INTERFACE I_EventGroupItem

METHOD PUBLIC AddHandler
VAR_INPUT
	EventHandler : I_EventHandler;
END_VAR
END_METHOD

METHOD PUBLIC Dispose
VAR_INPUT
END_VAR
END_METHOD

METHOD PUBLIC Emit
VAR_INPUT
	Event : I_Event;
END_VAR
END_METHOD

METHOD EqualTo : BOOL
VAR_INPUT
	Name : T_MAXSTRING;
END_VAR
END_METHOD

PROPERTY HasHandlers : BOOL
GET
END_GET
END_PROPERTY

PROPERTY PUBLIC Next : I_EventGroupItem
GET
END_GET
SET
END_SET
END_PROPERTY

PROPERTY PUBLIC Previous : I_EventGroupItem
GET
END_GET
SET
END_SET
END_PROPERTY

METHOD RemoveHandler
VAR_INPUT
	EventHandler : I_EventHandler;
END_VAR
END_METHOD

END_INTERFACE

(* stored: Version 1.1.0.1, ProductVersion 3.1.4024.12
   Itf I_EventGroupItem: Id {7a1aa493-2557-41cb-abb3-c16bd9197aae}
   Method AddHandler: Id {23b0f7b4-8051-4dc6-b2fb-d9f1a5f6af37}
   Method Dispose: Id {1d9a84c7-e06c-4aa0-b10a-8120bf170ab4}
   Method Emit: Id {057fcb02-01ee-4f3e-b199-c01963cdefe8}
   Method EqualTo: Id {a0733ef6-95ca-4a6b-b85f-8b85d11ec1e1}
   Property HasHandlers: Id {1d0156d6-948d-4c09-9e8c-940fdf299838}
   Get Get: Id {f93f0960-7100-4f32-804b-08f516727210}
   Property Next: Id {9f8ae168-7fea-40e1-8194-bd7be4b40641}
   Get Get: Id {b1fb12e4-77d8-403f-b6bc-1a0b71d27fdb}
   Set Set: Id {e75730ee-4035-400f-b60a-402a8c222263}
   Property Previous: Id {5146e2bd-74bf-4f34-85d5-27a83b3bda15}
   Get Get: Id {8fa99a83-f4b3-41ba-8c3b-85d444170eb1}
   Set Set: Id {016751a6-3dd7-4502-9a9d-3efd996d0cad}
   Method RemoveHandler: Id {a14327f5-d797-4e0f-9ccb-a6bc2e8ca8ef} *)
